DATA_BLOCK "DB_MachineConfig"
{ S7_Optimized_Access := 'TRUE' }
VERSION : 0.1
NON_RETAIN
   VAR
      lastError : Int;
      lastErrorBrand : Int;
      brand { S7_SetPoint := 'False'} : Array[1..16] of "UDT_MachineIOConfig";
   END_VAR


BEGIN
   lastError := 201;
   lastErrorBrand := 2;
   brand[1]."name" := 'Spinner';
   brand[1].cycleArchetype := 1;
   brand[1].in[0].present := TRUE;
   brand[1].in[0].byteOff := 0;
   brand[1].in[0].bitOff := 0;
   brand[1].in[0].inverted := FALSE;
   brand[1].in[1].present := FALSE;
   brand[1].in[1].byteOff := 0;
   brand[1].in[1].bitOff := 0;
   brand[1].in[1].inverted := FALSE;
   brand[1].in[2].present := TRUE;
   brand[1].in[2].byteOff := 0;
   brand[1].in[2].bitOff := 1;
   brand[1].in[2].inverted := FALSE;
   brand[1].in[3].present := TRUE;
   brand[1].in[3].byteOff := 0;
   brand[1].in[3].bitOff := 2;
   brand[1].in[3].inverted := FALSE;
   brand[1].in[4].present := TRUE;
   brand[1].in[4].byteOff := 0;
   brand[1].in[4].bitOff := 3;
   brand[1].in[4].inverted := FALSE;
   brand[1].in[5].present := FALSE;
   brand[1].in[5].byteOff := 0;
   brand[1].in[5].bitOff := 0;
   brand[1].in[5].inverted := FALSE;
   brand[1].in[6].present := TRUE;
   brand[1].in[6].byteOff := 0;
   brand[1].in[6].bitOff := 4;
   brand[1].in[6].inverted := FALSE;
   brand[1].in[7].present := TRUE;
   brand[1].in[7].byteOff := 0;
   brand[1].in[7].bitOff := 5;
   brand[1].in[7].inverted := FALSE;
   brand[1].in[8].present := TRUE;
   brand[1].in[8].byteOff := 0;
   brand[1].in[8].bitOff := 6;
   brand[1].in[8].inverted := FALSE;
   brand[1].in[9].present := FALSE;
   brand[1].in[9].byteOff := 0;
   brand[1].in[9].bitOff := 0;
   brand[1].in[9].inverted := FALSE;
   brand[1].out[0].present := TRUE;
   brand[1].out[0].byteOff := 0;
   brand[1].out[0].bitOff := 0;
   brand[1].out[0].inverted := FALSE;
   brand[1].out[1].present := FALSE;
   brand[1].out[1].byteOff := 0;
   brand[1].out[1].bitOff := 0;
   brand[1].out[1].inverted := FALSE;
   brand[1].out[2].present := TRUE;
   brand[1].out[2].byteOff := 0;
   brand[1].out[2].bitOff := 1;
   brand[1].out[2].inverted := FALSE;
   brand[1].out[3].present := TRUE;
   brand[1].out[3].byteOff := 0;
   brand[1].out[3].bitOff := 2;
   brand[1].out[3].inverted := FALSE;
   brand[1].out[4].present := TRUE;
   brand[1].out[4].byteOff := 0;
   brand[1].out[4].bitOff := 3;
   brand[1].out[4].inverted := FALSE;
   brand[1].out[5].present := FALSE;
   brand[1].out[5].byteOff := 0;
   brand[1].out[5].bitOff := 0;
   brand[1].out[5].inverted := FALSE;
   brand[1].out[6].present := FALSE;
   brand[1].out[6].byteOff := 0;
   brand[1].out[6].bitOff := 0;
   brand[1].out[6].inverted := FALSE;
   brand[1].out[7].present := FALSE;
   brand[1].out[7].byteOff := 0;
   brand[1].out[7].bitOff := 0;
   brand[1].out[7].inverted := FALSE;
   brand[1].out[8].present := TRUE;
   brand[1].out[8].byteOff := 0;
   brand[1].out[8].bitOff := 4;
   brand[1].out[8].inverted := FALSE;
   brand[1].out[9].present := TRUE;
   brand[1].out[9].byteOff := 0;
   brand[1].out[9].bitOff := 5;
   brand[1].out[9].inverted := FALSE;
   brand[1].out[10].present := FALSE;
   brand[1].out[10].byteOff := 0;
   brand[1].out[10].bitOff := 0;
   brand[1].out[10].inverted := FALSE;
   brand[2]."name" := 'HAAS';
   brand[2].cycleArchetype := 2;
   brand[2].in[0].present := TRUE;
   brand[2].in[0].byteOff := 0;
   brand[2].in[0].bitOff := 2;
   brand[2].in[0].inverted := TRUE;
   brand[2].in[1].present := TRUE;
   brand[2].in[1].byteOff := 0;
   brand[2].in[1].bitOff := 2;
   brand[2].in[1].inverted := FALSE;
   brand[2].in[2].present := TRUE;
   brand[2].in[2].byteOff := 0;
   brand[2].in[2].bitOff := 4;
   brand[2].in[2].inverted := FALSE;
   brand[2].in[3].present := TRUE;
   brand[2].in[3].byteOff := 0;
   brand[2].in[3].bitOff := 5;
   brand[2].in[3].inverted := FALSE;
   brand[2].in[4].present := TRUE;
   brand[2].in[4].byteOff := 0;
   brand[2].in[4].bitOff := 6;
   brand[2].in[4].inverted := FALSE;
   brand[2].in[5].present := TRUE;
   brand[2].in[5].byteOff := 0;
   brand[2].in[5].bitOff := 7;
   brand[2].in[5].inverted := FALSE;
   brand[2].in[6].present := TRUE;
   brand[2].in[6].byteOff := 0;
   brand[2].in[6].bitOff := 0;
   brand[2].in[6].inverted := FALSE;
   brand[2].in[7].present := TRUE;
   brand[2].in[7].byteOff := 0;
   brand[2].in[7].bitOff := 1;
   brand[2].in[7].inverted := FALSE;
   brand[2].in[8].present := FALSE;
   brand[2].in[8].byteOff := 0;
   brand[2].in[8].bitOff := 0;
   brand[2].in[8].inverted := FALSE;
   brand[2].in[9].present := FALSE;
   brand[2].in[9].byteOff := 0;
   brand[2].in[9].bitOff := 0;
   brand[2].in[9].inverted := FALSE;
   brand[2].out[0].present := FALSE;
   brand[2].out[0].byteOff := 0;
   brand[2].out[0].bitOff := 0;
   brand[2].out[0].inverted := FALSE;
   brand[2].out[1].present := FALSE;
   brand[2].out[1].byteOff := 0;
   brand[2].out[1].bitOff := 0;
   brand[2].out[1].inverted := FALSE;
   brand[2].out[2].present := TRUE;
   brand[2].out[2].byteOff := 0;
   brand[2].out[2].bitOff := 2;
   brand[2].out[2].inverted := FALSE;
   brand[2].out[3].present := TRUE;
   brand[2].out[3].byteOff := 0;
   brand[2].out[3].bitOff := 3;
   brand[2].out[3].inverted := FALSE;
   brand[2].out[4].present := TRUE;
   brand[2].out[4].byteOff := 0;
   brand[2].out[4].bitOff := 4;
   brand[2].out[4].inverted := FALSE;
   brand[2].out[5].present := TRUE;
   brand[2].out[5].byteOff := 0;
   brand[2].out[5].bitOff := 5;
   brand[2].out[5].inverted := FALSE;
   brand[2].out[6].present := FALSE;
   brand[2].out[6].byteOff := 0;
   brand[2].out[6].bitOff := 0;
   brand[2].out[6].inverted := FALSE;
   brand[2].out[7].present := FALSE;
   brand[2].out[7].byteOff := 0;
   brand[2].out[7].bitOff := 0;
   brand[2].out[7].inverted := FALSE;
   brand[2].out[8].present := TRUE;
   brand[2].out[8].byteOff := 0;
   brand[2].out[8].bitOff := 0;
   brand[2].out[8].inverted := FALSE;
   brand[2].out[9].present := TRUE;
   brand[2].out[9].byteOff := 0;
   brand[2].out[9].bitOff := 6;
   brand[2].out[9].inverted := FALSE;
   brand[2].out[10].present := TRUE;
   brand[2].out[10].byteOff := 0;
   brand[2].out[10].bitOff := 1;
   brand[2].out[10].inverted := FALSE;
   brand[3]."name" := '';
   brand[3].cycleArchetype := 0;
   brand[3].in[0].present := FALSE;
   brand[3].in[0].byteOff := 0;
   brand[3].in[0].bitOff := 0;
   brand[3].in[0].inverted := FALSE;
   brand[3].in[1].present := FALSE;
   brand[3].in[1].byteOff := 0;
   brand[3].in[1].bitOff := 0;
   brand[3].in[1].inverted := FALSE;
   brand[3].in[2].present := FALSE;
   brand[3].in[2].byteOff := 0;
   brand[3].in[2].bitOff := 0;
   brand[3].in[2].inverted := FALSE;
   brand[3].in[3].present := FALSE;
   brand[3].in[3].byteOff := 0;
   brand[3].in[3].bitOff := 0;
   brand[3].in[3].inverted := FALSE;
   brand[3].in[4].present := FALSE;
   brand[3].in[4].byteOff := 0;
   brand[3].in[4].bitOff := 0;
   brand[3].in[4].inverted := FALSE;
   brand[3].in[5].present := FALSE;
   brand[3].in[5].byteOff := 0;
   brand[3].in[5].bitOff := 0;
   brand[3].in[5].inverted := FALSE;
   brand[3].in[6].present := FALSE;
   brand[3].in[6].byteOff := 0;
   brand[3].in[6].bitOff := 0;
   brand[3].in[6].inverted := FALSE;
   brand[3].in[7].present := FALSE;
   brand[3].in[7].byteOff := 0;
   brand[3].in[7].bitOff := 0;
   brand[3].in[7].inverted := FALSE;
   brand[3].in[8].present := FALSE;
   brand[3].in[8].byteOff := 0;
   brand[3].in[8].bitOff := 0;
   brand[3].in[8].inverted := FALSE;
   brand[3].in[9].present := FALSE;
   brand[3].in[9].byteOff := 0;
   brand[3].in[9].bitOff := 0;
   brand[3].in[9].inverted := FALSE;
   brand[3].out[0].present := FALSE;
   brand[3].out[0].byteOff := 0;
   brand[3].out[0].bitOff := 0;
   brand[3].out[0].inverted := FALSE;
   brand[3].out[1].present := FALSE;
   brand[3].out[1].byteOff := 0;
   brand[3].out[1].bitOff := 0;
   brand[3].out[1].inverted := FALSE;
   brand[3].out[2].present := FALSE;
   brand[3].out[2].byteOff := 0;
   brand[3].out[2].bitOff := 0;
   brand[3].out[2].inverted := FALSE;
   brand[3].out[3].present := FALSE;
   brand[3].out[3].byteOff := 0;
   brand[3].out[3].bitOff := 0;
   brand[3].out[3].inverted := FALSE;
   brand[3].out[4].present := FALSE;
   brand[3].out[4].byteOff := 0;
   brand[3].out[4].bitOff := 0;
   brand[3].out[4].inverted := FALSE;
   brand[3].out[5].present := FALSE;
   brand[3].out[5].byteOff := 0;
   brand[3].out[5].bitOff := 0;
   brand[3].out[5].inverted := FALSE;
   brand[3].out[6].present := FALSE;
   brand[3].out[6].byteOff := 0;
   brand[3].out[6].bitOff := 0;
   brand[3].out[6].inverted := FALSE;
   brand[3].out[7].present := FALSE;
   brand[3].out[7].byteOff := 0;
   brand[3].out[7].bitOff := 0;
   brand[3].out[7].inverted := FALSE;
   brand[3].out[8].present := FALSE;
   brand[3].out[8].byteOff := 0;
   brand[3].out[8].bitOff := 0;
   brand[3].out[8].inverted := FALSE;
   brand[3].out[9].present := FALSE;
   brand[3].out[9].byteOff := 0;
   brand[3].out[9].bitOff := 0;
   brand[3].out[9].inverted := FALSE;
   brand[3].out[10].present := FALSE;
   brand[3].out[10].byteOff := 0;
   brand[3].out[10].bitOff := 0;
   brand[3].out[10].inverted := FALSE;
   brand[4]."name" := '';
   brand[4].cycleArchetype := 0;
   brand[4].in[0].present := FALSE;
   brand[4].in[0].byteOff := 0;
   brand[4].in[0].bitOff := 0;
   brand[4].in[0].inverted := FALSE;
   brand[4].in[1].present := FALSE;
   brand[4].in[1].byteOff := 0;
   brand[4].in[1].bitOff := 0;
   brand[4].in[1].inverted := FALSE;
   brand[4].in[2].present := FALSE;
   brand[4].in[2].byteOff := 0;
   brand[4].in[2].bitOff := 0;
   brand[4].in[2].inverted := FALSE;
   brand[4].in[3].present := FALSE;
   brand[4].in[3].byteOff := 0;
   brand[4].in[3].bitOff := 0;
   brand[4].in[3].inverted := FALSE;
   brand[4].in[4].present := FALSE;
   brand[4].in[4].byteOff := 0;
   brand[4].in[4].bitOff := 0;
   brand[4].in[4].inverted := FALSE;
   brand[4].in[5].present := FALSE;
   brand[4].in[5].byteOff := 0;
   brand[4].in[5].bitOff := 0;
   brand[4].in[5].inverted := FALSE;
   brand[4].in[6].present := FALSE;
   brand[4].in[6].byteOff := 0;
   brand[4].in[6].bitOff := 0;
   brand[4].in[6].inverted := FALSE;
   brand[4].in[7].present := FALSE;
   brand[4].in[7].byteOff := 0;
   brand[4].in[7].bitOff := 0;
   brand[4].in[7].inverted := FALSE;
   brand[4].in[8].present := FALSE;
   brand[4].in[8].byteOff := 0;
   brand[4].in[8].bitOff := 0;
   brand[4].in[8].inverted := FALSE;
   brand[4].in[9].present := FALSE;
   brand[4].in[9].byteOff := 0;
   brand[4].in[9].bitOff := 0;
   brand[4].in[9].inverted := FALSE;
   brand[4].out[0].present := FALSE;
   brand[4].out[0].byteOff := 0;
   brand[4].out[0].bitOff := 0;
   brand[4].out[0].inverted := FALSE;
   brand[4].out[1].present := FALSE;
   brand[4].out[1].byteOff := 0;
   brand[4].out[1].bitOff := 0;
   brand[4].out[1].inverted := FALSE;
   brand[4].out[2].present := FALSE;
   brand[4].out[2].byteOff := 0;
   brand[4].out[2].bitOff := 0;
   brand[4].out[2].inverted := FALSE;
   brand[4].out[3].present := FALSE;
   brand[4].out[3].byteOff := 0;
   brand[4].out[3].bitOff := 0;
   brand[4].out[3].inverted := FALSE;
   brand[4].out[4].present := FALSE;
   brand[4].out[4].byteOff := 0;
   brand[4].out[4].bitOff := 0;
   brand[4].out[4].inverted := FALSE;
   brand[4].out[5].present := FALSE;
   brand[4].out[5].byteOff := 0;
   brand[4].out[5].bitOff := 0;
   brand[4].out[5].inverted := FALSE;
   brand[4].out[6].present := FALSE;
   brand[4].out[6].byteOff := 0;
   brand[4].out[6].bitOff := 0;
   brand[4].out[6].inverted := FALSE;
   brand[4].out[7].present := FALSE;
   brand[4].out[7].byteOff := 0;
   brand[4].out[7].bitOff := 0;
   brand[4].out[7].inverted := FALSE;
   brand[4].out[8].present := FALSE;
   brand[4].out[8].byteOff := 0;
   brand[4].out[8].bitOff := 0;
   brand[4].out[8].inverted := FALSE;
   brand[4].out[9].present := FALSE;
   brand[4].out[9].byteOff := 0;
   brand[4].out[9].bitOff := 0;
   brand[4].out[9].inverted := FALSE;
   brand[4].out[10].present := FALSE;
   brand[4].out[10].byteOff := 0;
   brand[4].out[10].bitOff := 0;
   brand[4].out[10].inverted := FALSE;
   brand[5]."name" := '';
   brand[5].cycleArchetype := 0;
   brand[5].in[0].present := FALSE;
   brand[5].in[0].byteOff := 0;
   brand[5].in[0].bitOff := 0;
   brand[5].in[0].inverted := FALSE;
   brand[5].in[1].present := FALSE;
   brand[5].in[1].byteOff := 0;
   brand[5].in[1].bitOff := 0;
   brand[5].in[1].inverted := FALSE;
   brand[5].in[2].present := FALSE;
   brand[5].in[2].byteOff := 0;
   brand[5].in[2].bitOff := 0;
   brand[5].in[2].inverted := FALSE;
   brand[5].in[3].present := FALSE;
   brand[5].in[3].byteOff := 0;
   brand[5].in[3].bitOff := 0;
   brand[5].in[3].inverted := FALSE;
   brand[5].in[4].present := FALSE;
   brand[5].in[4].byteOff := 0;
   brand[5].in[4].bitOff := 0;
   brand[5].in[4].inverted := FALSE;
   brand[5].in[5].present := FALSE;
   brand[5].in[5].byteOff := 0;
   brand[5].in[5].bitOff := 0;
   brand[5].in[5].inverted := FALSE;
   brand[5].in[6].present := FALSE;
   brand[5].in[6].byteOff := 0;
   brand[5].in[6].bitOff := 0;
   brand[5].in[6].inverted := FALSE;
   brand[5].in[7].present := FALSE;
   brand[5].in[7].byteOff := 0;
   brand[5].in[7].bitOff := 0;
   brand[5].in[7].inverted := FALSE;
   brand[5].in[8].present := FALSE;
   brand[5].in[8].byteOff := 0;
   brand[5].in[8].bitOff := 0;
   brand[5].in[8].inverted := FALSE;
   brand[5].in[9].present := FALSE;
   brand[5].in[9].byteOff := 0;
   brand[5].in[9].bitOff := 0;
   brand[5].in[9].inverted := FALSE;
   brand[5].out[0].present := FALSE;
   brand[5].out[0].byteOff := 0;
   brand[5].out[0].bitOff := 0;
   brand[5].out[0].inverted := FALSE;
   brand[5].out[1].present := FALSE;
   brand[5].out[1].byteOff := 0;
   brand[5].out[1].bitOff := 0;
   brand[5].out[1].inverted := FALSE;
   brand[5].out[2].present := FALSE;
   brand[5].out[2].byteOff := 0;
   brand[5].out[2].bitOff := 0;
   brand[5].out[2].inverted := FALSE;
   brand[5].out[3].present := FALSE;
   brand[5].out[3].byteOff := 0;
   brand[5].out[3].bitOff := 0;
   brand[5].out[3].inverted := FALSE;
   brand[5].out[4].present := FALSE;
   brand[5].out[4].byteOff := 0;
   brand[5].out[4].bitOff := 0;
   brand[5].out[4].inverted := FALSE;
   brand[5].out[5].present := FALSE;
   brand[5].out[5].byteOff := 0;
   brand[5].out[5].bitOff := 0;
   brand[5].out[5].inverted := FALSE;
   brand[5].out[6].present := FALSE;
   brand[5].out[6].byteOff := 0;
   brand[5].out[6].bitOff := 0;
   brand[5].out[6].inverted := FALSE;
   brand[5].out[7].present := FALSE;
   brand[5].out[7].byteOff := 0;
   brand[5].out[7].bitOff := 0;
   brand[5].out[7].inverted := FALSE;
   brand[5].out[8].present := FALSE;
   brand[5].out[8].byteOff := 0;
   brand[5].out[8].bitOff := 0;
   brand[5].out[8].inverted := FALSE;
   brand[5].out[9].present := FALSE;
   brand[5].out[9].byteOff := 0;
   brand[5].out[9].bitOff := 0;
   brand[5].out[9].inverted := FALSE;
   brand[5].out[10].present := FALSE;
   brand[5].out[10].byteOff := 0;
   brand[5].out[10].bitOff := 0;
   brand[5].out[10].inverted := FALSE;
   brand[6]."name" := '';
   brand[6].cycleArchetype := 0;
   brand[6].in[0].present := FALSE;
   brand[6].in[0].byteOff := 0;
   brand[6].in[0].bitOff := 0;
   brand[6].in[0].inverted := FALSE;
   brand[6].in[1].present := FALSE;
   brand[6].in[1].byteOff := 0;
   brand[6].in[1].bitOff := 0;
   brand[6].in[1].inverted := FALSE;
   brand[6].in[2].present := FALSE;
   brand[6].in[2].byteOff := 0;
   brand[6].in[2].bitOff := 0;
   brand[6].in[2].inverted := FALSE;
   brand[6].in[3].present := FALSE;
   brand[6].in[3].byteOff := 0;
   brand[6].in[3].bitOff := 0;
   brand[6].in[3].inverted := FALSE;
   brand[6].in[4].present := FALSE;
   brand[6].in[4].byteOff := 0;
   brand[6].in[4].bitOff := 0;
   brand[6].in[4].inverted := FALSE;
   brand[6].in[5].present := FALSE;
   brand[6].in[5].byteOff := 0;
   brand[6].in[5].bitOff := 0;
   brand[6].in[5].inverted := FALSE;
   brand[6].in[6].present := FALSE;
   brand[6].in[6].byteOff := 0;
   brand[6].in[6].bitOff := 0;
   brand[6].in[6].inverted := FALSE;
   brand[6].in[7].present := FALSE;
   brand[6].in[7].byteOff := 0;
   brand[6].in[7].bitOff := 0;
   brand[6].in[7].inverted := FALSE;
   brand[6].in[8].present := FALSE;
   brand[6].in[8].byteOff := 0;
   brand[6].in[8].bitOff := 0;
   brand[6].in[8].inverted := FALSE;
   brand[6].in[9].present := FALSE;
   brand[6].in[9].byteOff := 0;
   brand[6].in[9].bitOff := 0;
   brand[6].in[9].inverted := FALSE;
   brand[6].out[0].present := FALSE;
   brand[6].out[0].byteOff := 0;
   brand[6].out[0].bitOff := 0;
   brand[6].out[0].inverted := FALSE;
   brand[6].out[1].present := FALSE;
   brand[6].out[1].byteOff := 0;
   brand[6].out[1].bitOff := 0;
   brand[6].out[1].inverted := FALSE;
   brand[6].out[2].present := FALSE;
   brand[6].out[2].byteOff := 0;
   brand[6].out[2].bitOff := 0;
   brand[6].out[2].inverted := FALSE;
   brand[6].out[3].present := FALSE;
   brand[6].out[3].byteOff := 0;
   brand[6].out[3].bitOff := 0;
   brand[6].out[3].inverted := FALSE;
   brand[6].out[4].present := FALSE;
   brand[6].out[4].byteOff := 0;
   brand[6].out[4].bitOff := 0;
   brand[6].out[4].inverted := FALSE;
   brand[6].out[5].present := FALSE;
   brand[6].out[5].byteOff := 0;
   brand[6].out[5].bitOff := 0;
   brand[6].out[5].inverted := FALSE;
   brand[6].out[6].present := FALSE;
   brand[6].out[6].byteOff := 0;
   brand[6].out[6].bitOff := 0;
   brand[6].out[6].inverted := FALSE;
   brand[6].out[7].present := FALSE;
   brand[6].out[7].byteOff := 0;
   brand[6].out[7].bitOff := 0;
   brand[6].out[7].inverted := FALSE;
   brand[6].out[8].present := FALSE;
   brand[6].out[8].byteOff := 0;
   brand[6].out[8].bitOff := 0;
   brand[6].out[8].inverted := FALSE;
   brand[6].out[9].present := FALSE;
   brand[6].out[9].byteOff := 0;
   brand[6].out[9].bitOff := 0;
   brand[6].out[9].inverted := FALSE;
   brand[6].out[10].present := FALSE;
   brand[6].out[10].byteOff := 0;
   brand[6].out[10].bitOff := 0;
   brand[6].out[10].inverted := FALSE;
   brand[7]."name" := '';
   brand[7].cycleArchetype := 0;
   brand[7].in[0].present := FALSE;
   brand[7].in[0].byteOff := 0;
   brand[7].in[0].bitOff := 0;
   brand[7].in[0].inverted := FALSE;
   brand[7].in[1].present := FALSE;
   brand[7].in[1].byteOff := 0;
   brand[7].in[1].bitOff := 0;
   brand[7].in[1].inverted := FALSE;
   brand[7].in[2].present := FALSE;
   brand[7].in[2].byteOff := 0;
   brand[7].in[2].bitOff := 0;
   brand[7].in[2].inverted := FALSE;
   brand[7].in[3].present := FALSE;
   brand[7].in[3].byteOff := 0;
   brand[7].in[3].bitOff := 0;
   brand[7].in[3].inverted := FALSE;
   brand[7].in[4].present := FALSE;
   brand[7].in[4].byteOff := 0;
   brand[7].in[4].bitOff := 0;
   brand[7].in[4].inverted := FALSE;
   brand[7].in[5].present := FALSE;
   brand[7].in[5].byteOff := 0;
   brand[7].in[5].bitOff := 0;
   brand[7].in[5].inverted := FALSE;
   brand[7].in[6].present := FALSE;
   brand[7].in[6].byteOff := 0;
   brand[7].in[6].bitOff := 0;
   brand[7].in[6].inverted := FALSE;
   brand[7].in[7].present := FALSE;
   brand[7].in[7].byteOff := 0;
   brand[7].in[7].bitOff := 0;
   brand[7].in[7].inverted := FALSE;
   brand[7].in[8].present := FALSE;
   brand[7].in[8].byteOff := 0;
   brand[7].in[8].bitOff := 0;
   brand[7].in[8].inverted := FALSE;
   brand[7].in[9].present := FALSE;
   brand[7].in[9].byteOff := 0;
   brand[7].in[9].bitOff := 0;
   brand[7].in[9].inverted := FALSE;
   brand[7].out[0].present := FALSE;
   brand[7].out[0].byteOff := 0;
   brand[7].out[0].bitOff := 0;
   brand[7].out[0].inverted := FALSE;
   brand[7].out[1].present := FALSE;
   brand[7].out[1].byteOff := 0;
   brand[7].out[1].bitOff := 0;
   brand[7].out[1].inverted := FALSE;
   brand[7].out[2].present := FALSE;
   brand[7].out[2].byteOff := 0;
   brand[7].out[2].bitOff := 0;
   brand[7].out[2].inverted := FALSE;
   brand[7].out[3].present := FALSE;
   brand[7].out[3].byteOff := 0;
   brand[7].out[3].bitOff := 0;
   brand[7].out[3].inverted := FALSE;
   brand[7].out[4].present := FALSE;
   brand[7].out[4].byteOff := 0;
   brand[7].out[4].bitOff := 0;
   brand[7].out[4].inverted := FALSE;
   brand[7].out[5].present := FALSE;
   brand[7].out[5].byteOff := 0;
   brand[7].out[5].bitOff := 0;
   brand[7].out[5].inverted := FALSE;
   brand[7].out[6].present := FALSE;
   brand[7].out[6].byteOff := 0;
   brand[7].out[6].bitOff := 0;
   brand[7].out[6].inverted := FALSE;
   brand[7].out[7].present := FALSE;
   brand[7].out[7].byteOff := 0;
   brand[7].out[7].bitOff := 0;
   brand[7].out[7].inverted := FALSE;
   brand[7].out[8].present := FALSE;
   brand[7].out[8].byteOff := 0;
   brand[7].out[8].bitOff := 0;
   brand[7].out[8].inverted := FALSE;
   brand[7].out[9].present := FALSE;
   brand[7].out[9].byteOff := 0;
   brand[7].out[9].bitOff := 0;
   brand[7].out[9].inverted := FALSE;
   brand[7].out[10].present := FALSE;
   brand[7].out[10].byteOff := 0;
   brand[7].out[10].bitOff := 0;
   brand[7].out[10].inverted := FALSE;
   brand[8]."name" := '';
   brand[8].cycleArchetype := 0;
   brand[8].in[0].present := FALSE;
   brand[8].in[0].byteOff := 0;
   brand[8].in[0].bitOff := 0;
   brand[8].in[0].inverted := FALSE;
   brand[8].in[1].present := FALSE;
   brand[8].in[1].byteOff := 0;
   brand[8].in[1].bitOff := 0;
   brand[8].in[1].inverted := FALSE;
   brand[8].in[2].present := FALSE;
   brand[8].in[2].byteOff := 0;
   brand[8].in[2].bitOff := 0;
   brand[8].in[2].inverted := FALSE;
   brand[8].in[3].present := FALSE;
   brand[8].in[3].byteOff := 0;
   brand[8].in[3].bitOff := 0;
   brand[8].in[3].inverted := FALSE;
   brand[8].in[4].present := FALSE;
   brand[8].in[4].byteOff := 0;
   brand[8].in[4].bitOff := 0;
   brand[8].in[4].inverted := FALSE;
   brand[8].in[5].present := FALSE;
   brand[8].in[5].byteOff := 0;
   brand[8].in[5].bitOff := 0;
   brand[8].in[5].inverted := FALSE;
   brand[8].in[6].present := FALSE;
   brand[8].in[6].byteOff := 0;
   brand[8].in[6].bitOff := 0;
   brand[8].in[6].inverted := FALSE;
   brand[8].in[7].present := FALSE;
   brand[8].in[7].byteOff := 0;
   brand[8].in[7].bitOff := 0;
   brand[8].in[7].inverted := FALSE;
   brand[8].in[8].present := FALSE;
   brand[8].in[8].byteOff := 0;
   brand[8].in[8].bitOff := 0;
   brand[8].in[8].inverted := FALSE;
   brand[8].in[9].present := FALSE;
   brand[8].in[9].byteOff := 0;
   brand[8].in[9].bitOff := 0;
   brand[8].in[9].inverted := FALSE;
   brand[8].out[0].present := FALSE;
   brand[8].out[0].byteOff := 0;
   brand[8].out[0].bitOff := 0;
   brand[8].out[0].inverted := FALSE;
   brand[8].out[1].present := FALSE;
   brand[8].out[1].byteOff := 0;
   brand[8].out[1].bitOff := 0;
   brand[8].out[1].inverted := FALSE;
   brand[8].out[2].present := FALSE;
   brand[8].out[2].byteOff := 0;
   brand[8].out[2].bitOff := 0;
   brand[8].out[2].inverted := FALSE;
   brand[8].out[3].present := FALSE;
   brand[8].out[3].byteOff := 0;
   brand[8].out[3].bitOff := 0;
   brand[8].out[3].inverted := FALSE;
   brand[8].out[4].present := FALSE;
   brand[8].out[4].byteOff := 0;
   brand[8].out[4].bitOff := 0;
   brand[8].out[4].inverted := FALSE;
   brand[8].out[5].present := FALSE;
   brand[8].out[5].byteOff := 0;
   brand[8].out[5].bitOff := 0;
   brand[8].out[5].inverted := FALSE;
   brand[8].out[6].present := FALSE;
   brand[8].out[6].byteOff := 0;
   brand[8].out[6].bitOff := 0;
   brand[8].out[6].inverted := FALSE;
   brand[8].out[7].present := FALSE;
   brand[8].out[7].byteOff := 0;
   brand[8].out[7].bitOff := 0;
   brand[8].out[7].inverted := FALSE;
   brand[8].out[8].present := FALSE;
   brand[8].out[8].byteOff := 0;
   brand[8].out[8].bitOff := 0;
   brand[8].out[8].inverted := FALSE;
   brand[8].out[9].present := FALSE;
   brand[8].out[9].byteOff := 0;
   brand[8].out[9].bitOff := 0;
   brand[8].out[9].inverted := FALSE;
   brand[8].out[10].present := FALSE;
   brand[8].out[10].byteOff := 0;
   brand[8].out[10].bitOff := 0;
   brand[8].out[10].inverted := FALSE;
   brand[9]."name" := '';
   brand[9].cycleArchetype := 0;
   brand[9].in[0].present := FALSE;
   brand[9].in[0].byteOff := 0;
   brand[9].in[0].bitOff := 0;
   brand[9].in[0].inverted := FALSE;
   brand[9].in[1].present := FALSE;
   brand[9].in[1].byteOff := 0;
   brand[9].in[1].bitOff := 0;
   brand[9].in[1].inverted := FALSE;
   brand[9].in[2].present := FALSE;
   brand[9].in[2].byteOff := 0;
   brand[9].in[2].bitOff := 0;
   brand[9].in[2].inverted := FALSE;
   brand[9].in[3].present := FALSE;
   brand[9].in[3].byteOff := 0;
   brand[9].in[3].bitOff := 0;
   brand[9].in[3].inverted := FALSE;
   brand[9].in[4].present := FALSE;
   brand[9].in[4].byteOff := 0;
   brand[9].in[4].bitOff := 0;
   brand[9].in[4].inverted := FALSE;
   brand[9].in[5].present := FALSE;
   brand[9].in[5].byteOff := 0;
   brand[9].in[5].bitOff := 0;
   brand[9].in[5].inverted := FALSE;
   brand[9].in[6].present := FALSE;
   brand[9].in[6].byteOff := 0;
   brand[9].in[6].bitOff := 0;
   brand[9].in[6].inverted := FALSE;
   brand[9].in[7].present := FALSE;
   brand[9].in[7].byteOff := 0;
   brand[9].in[7].bitOff := 0;
   brand[9].in[7].inverted := FALSE;
   brand[9].in[8].present := FALSE;
   brand[9].in[8].byteOff := 0;
   brand[9].in[8].bitOff := 0;
   brand[9].in[8].inverted := FALSE;
   brand[9].in[9].present := FALSE;
   brand[9].in[9].byteOff := 0;
   brand[9].in[9].bitOff := 0;
   brand[9].in[9].inverted := FALSE;
   brand[9].out[0].present := FALSE;
   brand[9].out[0].byteOff := 0;
   brand[9].out[0].bitOff := 0;
   brand[9].out[0].inverted := FALSE;
   brand[9].out[1].present := FALSE;
   brand[9].out[1].byteOff := 0;
   brand[9].out[1].bitOff := 0;
   brand[9].out[1].inverted := FALSE;
   brand[9].out[2].present := FALSE;
   brand[9].out[2].byteOff := 0;
   brand[9].out[2].bitOff := 0;
   brand[9].out[2].inverted := FALSE;
   brand[9].out[3].present := FALSE;
   brand[9].out[3].byteOff := 0;
   brand[9].out[3].bitOff := 0;
   brand[9].out[3].inverted := FALSE;
   brand[9].out[4].present := FALSE;
   brand[9].out[4].byteOff := 0;
   brand[9].out[4].bitOff := 0;
   brand[9].out[4].inverted := FALSE;
   brand[9].out[5].present := FALSE;
   brand[9].out[5].byteOff := 0;
   brand[9].out[5].bitOff := 0;
   brand[9].out[5].inverted := FALSE;
   brand[9].out[6].present := FALSE;
   brand[9].out[6].byteOff := 0;
   brand[9].out[6].bitOff := 0;
   brand[9].out[6].inverted := FALSE;
   brand[9].out[7].present := FALSE;
   brand[9].out[7].byteOff := 0;
   brand[9].out[7].bitOff := 0;
   brand[9].out[7].inverted := FALSE;
   brand[9].out[8].present := FALSE;
   brand[9].out[8].byteOff := 0;
   brand[9].out[8].bitOff := 0;
   brand[9].out[8].inverted := FALSE;
   brand[9].out[9].present := FALSE;
   brand[9].out[9].byteOff := 0;
   brand[9].out[9].bitOff := 0;
   brand[9].out[9].inverted := FALSE;
   brand[9].out[10].present := FALSE;
   brand[9].out[10].byteOff := 0;
   brand[9].out[10].bitOff := 0;
   brand[9].out[10].inverted := FALSE;
   brand[10]."name" := '';
   brand[10].cycleArchetype := 0;
   brand[10].in[0].present := FALSE;
   brand[10].in[0].byteOff := 0;
   brand[10].in[0].bitOff := 0;
   brand[10].in[0].inverted := FALSE;
   brand[10].in[1].present := FALSE;
   brand[10].in[1].byteOff := 0;
   brand[10].in[1].bitOff := 0;
   brand[10].in[1].inverted := FALSE;
   brand[10].in[2].present := FALSE;
   brand[10].in[2].byteOff := 0;
   brand[10].in[2].bitOff := 0;
   brand[10].in[2].inverted := FALSE;
   brand[10].in[3].present := FALSE;
   brand[10].in[3].byteOff := 0;
   brand[10].in[3].bitOff := 0;
   brand[10].in[3].inverted := FALSE;
   brand[10].in[4].present := FALSE;
   brand[10].in[4].byteOff := 0;
   brand[10].in[4].bitOff := 0;
   brand[10].in[4].inverted := FALSE;
   brand[10].in[5].present := FALSE;
   brand[10].in[5].byteOff := 0;
   brand[10].in[5].bitOff := 0;
   brand[10].in[5].inverted := FALSE;
   brand[10].in[6].present := FALSE;
   brand[10].in[6].byteOff := 0;
   brand[10].in[6].bitOff := 0;
   brand[10].in[6].inverted := FALSE;
   brand[10].in[7].present := FALSE;
   brand[10].in[7].byteOff := 0;
   brand[10].in[7].bitOff := 0;
   brand[10].in[7].inverted := FALSE;
   brand[10].in[8].present := FALSE;
   brand[10].in[8].byteOff := 0;
   brand[10].in[8].bitOff := 0;
   brand[10].in[8].inverted := FALSE;
   brand[10].in[9].present := FALSE;
   brand[10].in[9].byteOff := 0;
   brand[10].in[9].bitOff := 0;
   brand[10].in[9].inverted := FALSE;
   brand[10].out[0].present := FALSE;
   brand[10].out[0].byteOff := 0;
   brand[10].out[0].bitOff := 0;
   brand[10].out[0].inverted := FALSE;
   brand[10].out[1].present := FALSE;
   brand[10].out[1].byteOff := 0;
   brand[10].out[1].bitOff := 0;
   brand[10].out[1].inverted := FALSE;
   brand[10].out[2].present := FALSE;
   brand[10].out[2].byteOff := 0;
   brand[10].out[2].bitOff := 0;
   brand[10].out[2].inverted := FALSE;
   brand[10].out[3].present := FALSE;
   brand[10].out[3].byteOff := 0;
   brand[10].out[3].bitOff := 0;
   brand[10].out[3].inverted := FALSE;
   brand[10].out[4].present := FALSE;
   brand[10].out[4].byteOff := 0;
   brand[10].out[4].bitOff := 0;
   brand[10].out[4].inverted := FALSE;
   brand[10].out[5].present := FALSE;
   brand[10].out[5].byteOff := 0;
   brand[10].out[5].bitOff := 0;
   brand[10].out[5].inverted := FALSE;
   brand[10].out[6].present := FALSE;
   brand[10].out[6].byteOff := 0;
   brand[10].out[6].bitOff := 0;
   brand[10].out[6].inverted := FALSE;
   brand[10].out[7].present := FALSE;
   brand[10].out[7].byteOff := 0;
   brand[10].out[7].bitOff := 0;
   brand[10].out[7].inverted := FALSE;
   brand[10].out[8].present := FALSE;
   brand[10].out[8].byteOff := 0;
   brand[10].out[8].bitOff := 0;
   brand[10].out[8].inverted := FALSE;
   brand[10].out[9].present := FALSE;
   brand[10].out[9].byteOff := 0;
   brand[10].out[9].bitOff := 0;
   brand[10].out[9].inverted := FALSE;
   brand[10].out[10].present := FALSE;
   brand[10].out[10].byteOff := 0;
   brand[10].out[10].bitOff := 0;
   brand[10].out[10].inverted := FALSE;
   brand[11]."name" := '';
   brand[11].cycleArchetype := 0;
   brand[11].in[0].present := FALSE;
   brand[11].in[0].byteOff := 0;
   brand[11].in[0].bitOff := 0;
   brand[11].in[0].inverted := FALSE;
   brand[11].in[1].present := FALSE;
   brand[11].in[1].byteOff := 0;
   brand[11].in[1].bitOff := 0;
   brand[11].in[1].inverted := FALSE;
   brand[11].in[2].present := FALSE;
   brand[11].in[2].byteOff := 0;
   brand[11].in[2].bitOff := 0;
   brand[11].in[2].inverted := FALSE;
   brand[11].in[3].present := FALSE;
   brand[11].in[3].byteOff := 0;
   brand[11].in[3].bitOff := 0;
   brand[11].in[3].inverted := FALSE;
   brand[11].in[4].present := FALSE;
   brand[11].in[4].byteOff := 0;
   brand[11].in[4].bitOff := 0;
   brand[11].in[4].inverted := FALSE;
   brand[11].in[5].present := FALSE;
   brand[11].in[5].byteOff := 0;
   brand[11].in[5].bitOff := 0;
   brand[11].in[5].inverted := FALSE;
   brand[11].in[6].present := FALSE;
   brand[11].in[6].byteOff := 0;
   brand[11].in[6].bitOff := 0;
   brand[11].in[6].inverted := FALSE;
   brand[11].in[7].present := FALSE;
   brand[11].in[7].byteOff := 0;
   brand[11].in[7].bitOff := 0;
   brand[11].in[7].inverted := FALSE;
   brand[11].in[8].present := FALSE;
   brand[11].in[8].byteOff := 0;
   brand[11].in[8].bitOff := 0;
   brand[11].in[8].inverted := FALSE;
   brand[11].in[9].present := FALSE;
   brand[11].in[9].byteOff := 0;
   brand[11].in[9].bitOff := 0;
   brand[11].in[9].inverted := FALSE;
   brand[11].out[0].present := FALSE;
   brand[11].out[0].byteOff := 0;
   brand[11].out[0].bitOff := 0;
   brand[11].out[0].inverted := FALSE;
   brand[11].out[1].present := FALSE;
   brand[11].out[1].byteOff := 0;
   brand[11].out[1].bitOff := 0;
   brand[11].out[1].inverted := FALSE;
   brand[11].out[2].present := FALSE;
   brand[11].out[2].byteOff := 0;
   brand[11].out[2].bitOff := 0;
   brand[11].out[2].inverted := FALSE;
   brand[11].out[3].present := FALSE;
   brand[11].out[3].byteOff := 0;
   brand[11].out[3].bitOff := 0;
   brand[11].out[3].inverted := FALSE;
   brand[11].out[4].present := FALSE;
   brand[11].out[4].byteOff := 0;
   brand[11].out[4].bitOff := 0;
   brand[11].out[4].inverted := FALSE;
   brand[11].out[5].present := FALSE;
   brand[11].out[5].byteOff := 0;
   brand[11].out[5].bitOff := 0;
   brand[11].out[5].inverted := FALSE;
   brand[11].out[6].present := FALSE;
   brand[11].out[6].byteOff := 0;
   brand[11].out[6].bitOff := 0;
   brand[11].out[6].inverted := FALSE;
   brand[11].out[7].present := FALSE;
   brand[11].out[7].byteOff := 0;
   brand[11].out[7].bitOff := 0;
   brand[11].out[7].inverted := FALSE;
   brand[11].out[8].present := FALSE;
   brand[11].out[8].byteOff := 0;
   brand[11].out[8].bitOff := 0;
   brand[11].out[8].inverted := FALSE;
   brand[11].out[9].present := FALSE;
   brand[11].out[9].byteOff := 0;
   brand[11].out[9].bitOff := 0;
   brand[11].out[9].inverted := FALSE;
   brand[11].out[10].present := FALSE;
   brand[11].out[10].byteOff := 0;
   brand[11].out[10].bitOff := 0;
   brand[11].out[10].inverted := FALSE;
   brand[12]."name" := '';
   brand[12].cycleArchetype := 0;
   brand[12].in[0].present := FALSE;
   brand[12].in[0].byteOff := 0;
   brand[12].in[0].bitOff := 0;
   brand[12].in[0].inverted := FALSE;
   brand[12].in[1].present := FALSE;
   brand[12].in[1].byteOff := 0;
   brand[12].in[1].bitOff := 0;
   brand[12].in[1].inverted := FALSE;
   brand[12].in[2].present := FALSE;
   brand[12].in[2].byteOff := 0;
   brand[12].in[2].bitOff := 0;
   brand[12].in[2].inverted := FALSE;
   brand[12].in[3].present := FALSE;
   brand[12].in[3].byteOff := 0;
   brand[12].in[3].bitOff := 0;
   brand[12].in[3].inverted := FALSE;
   brand[12].in[4].present := FALSE;
   brand[12].in[4].byteOff := 0;
   brand[12].in[4].bitOff := 0;
   brand[12].in[4].inverted := FALSE;
   brand[12].in[5].present := FALSE;
   brand[12].in[5].byteOff := 0;
   brand[12].in[5].bitOff := 0;
   brand[12].in[5].inverted := FALSE;
   brand[12].in[6].present := FALSE;
   brand[12].in[6].byteOff := 0;
   brand[12].in[6].bitOff := 0;
   brand[12].in[6].inverted := FALSE;
   brand[12].in[7].present := FALSE;
   brand[12].in[7].byteOff := 0;
   brand[12].in[7].bitOff := 0;
   brand[12].in[7].inverted := FALSE;
   brand[12].in[8].present := FALSE;
   brand[12].in[8].byteOff := 0;
   brand[12].in[8].bitOff := 0;
   brand[12].in[8].inverted := FALSE;
   brand[12].in[9].present := FALSE;
   brand[12].in[9].byteOff := 0;
   brand[12].in[9].bitOff := 0;
   brand[12].in[9].inverted := FALSE;
   brand[12].out[0].present := FALSE;
   brand[12].out[0].byteOff := 0;
   brand[12].out[0].bitOff := 0;
   brand[12].out[0].inverted := FALSE;
   brand[12].out[1].present := FALSE;
   brand[12].out[1].byteOff := 0;
   brand[12].out[1].bitOff := 0;
   brand[12].out[1].inverted := FALSE;
   brand[12].out[2].present := FALSE;
   brand[12].out[2].byteOff := 0;
   brand[12].out[2].bitOff := 0;
   brand[12].out[2].inverted := FALSE;
   brand[12].out[3].present := FALSE;
   brand[12].out[3].byteOff := 0;
   brand[12].out[3].bitOff := 0;
   brand[12].out[3].inverted := FALSE;
   brand[12].out[4].present := FALSE;
   brand[12].out[4].byteOff := 0;
   brand[12].out[4].bitOff := 0;
   brand[12].out[4].inverted := FALSE;
   brand[12].out[5].present := FALSE;
   brand[12].out[5].byteOff := 0;
   brand[12].out[5].bitOff := 0;
   brand[12].out[5].inverted := FALSE;
   brand[12].out[6].present := FALSE;
   brand[12].out[6].byteOff := 0;
   brand[12].out[6].bitOff := 0;
   brand[12].out[6].inverted := FALSE;
   brand[12].out[7].present := FALSE;
   brand[12].out[7].byteOff := 0;
   brand[12].out[7].bitOff := 0;
   brand[12].out[7].inverted := FALSE;
   brand[12].out[8].present := FALSE;
   brand[12].out[8].byteOff := 0;
   brand[12].out[8].bitOff := 0;
   brand[12].out[8].inverted := FALSE;
   brand[12].out[9].present := FALSE;
   brand[12].out[9].byteOff := 0;
   brand[12].out[9].bitOff := 0;
   brand[12].out[9].inverted := FALSE;
   brand[12].out[10].present := FALSE;
   brand[12].out[10].byteOff := 0;
   brand[12].out[10].bitOff := 0;
   brand[12].out[10].inverted := FALSE;
   brand[13]."name" := '';
   brand[13].cycleArchetype := 0;
   brand[13].in[0].present := FALSE;
   brand[13].in[0].byteOff := 0;
   brand[13].in[0].bitOff := 0;
   brand[13].in[0].inverted := FALSE;
   brand[13].in[1].present := FALSE;
   brand[13].in[1].byteOff := 0;
   brand[13].in[1].bitOff := 0;
   brand[13].in[1].inverted := FALSE;
   brand[13].in[2].present := FALSE;
   brand[13].in[2].byteOff := 0;
   brand[13].in[2].bitOff := 0;
   brand[13].in[2].inverted := FALSE;
   brand[13].in[3].present := FALSE;
   brand[13].in[3].byteOff := 0;
   brand[13].in[3].bitOff := 0;
   brand[13].in[3].inverted := FALSE;
   brand[13].in[4].present := FALSE;
   brand[13].in[4].byteOff := 0;
   brand[13].in[4].bitOff := 0;
   brand[13].in[4].inverted := FALSE;
   brand[13].in[5].present := FALSE;
   brand[13].in[5].byteOff := 0;
   brand[13].in[5].bitOff := 0;
   brand[13].in[5].inverted := FALSE;
   brand[13].in[6].present := FALSE;
   brand[13].in[6].byteOff := 0;
   brand[13].in[6].bitOff := 0;
   brand[13].in[6].inverted := FALSE;
   brand[13].in[7].present := FALSE;
   brand[13].in[7].byteOff := 0;
   brand[13].in[7].bitOff := 0;
   brand[13].in[7].inverted := FALSE;
   brand[13].in[8].present := FALSE;
   brand[13].in[8].byteOff := 0;
   brand[13].in[8].bitOff := 0;
   brand[13].in[8].inverted := FALSE;
   brand[13].in[9].present := FALSE;
   brand[13].in[9].byteOff := 0;
   brand[13].in[9].bitOff := 0;
   brand[13].in[9].inverted := FALSE;
   brand[13].out[0].present := FALSE;
   brand[13].out[0].byteOff := 0;
   brand[13].out[0].bitOff := 0;
   brand[13].out[0].inverted := FALSE;
   brand[13].out[1].present := FALSE;
   brand[13].out[1].byteOff := 0;
   brand[13].out[1].bitOff := 0;
   brand[13].out[1].inverted := FALSE;
   brand[13].out[2].present := FALSE;
   brand[13].out[2].byteOff := 0;
   brand[13].out[2].bitOff := 0;
   brand[13].out[2].inverted := FALSE;
   brand[13].out[3].present := FALSE;
   brand[13].out[3].byteOff := 0;
   brand[13].out[3].bitOff := 0;
   brand[13].out[3].inverted := FALSE;
   brand[13].out[4].present := FALSE;
   brand[13].out[4].byteOff := 0;
   brand[13].out[4].bitOff := 0;
   brand[13].out[4].inverted := FALSE;
   brand[13].out[5].present := FALSE;
   brand[13].out[5].byteOff := 0;
   brand[13].out[5].bitOff := 0;
   brand[13].out[5].inverted := FALSE;
   brand[13].out[6].present := FALSE;
   brand[13].out[6].byteOff := 0;
   brand[13].out[6].bitOff := 0;
   brand[13].out[6].inverted := FALSE;
   brand[13].out[7].present := FALSE;
   brand[13].out[7].byteOff := 0;
   brand[13].out[7].bitOff := 0;
   brand[13].out[7].inverted := FALSE;
   brand[13].out[8].present := FALSE;
   brand[13].out[8].byteOff := 0;
   brand[13].out[8].bitOff := 0;
   brand[13].out[8].inverted := FALSE;
   brand[13].out[9].present := FALSE;
   brand[13].out[9].byteOff := 0;
   brand[13].out[9].bitOff := 0;
   brand[13].out[9].inverted := FALSE;
   brand[13].out[10].present := FALSE;
   brand[13].out[10].byteOff := 0;
   brand[13].out[10].bitOff := 0;
   brand[13].out[10].inverted := FALSE;
   brand[14]."name" := '';
   brand[14].cycleArchetype := 0;
   brand[14].in[0].present := FALSE;
   brand[14].in[0].byteOff := 0;
   brand[14].in[0].bitOff := 0;
   brand[14].in[0].inverted := FALSE;
   brand[14].in[1].present := FALSE;
   brand[14].in[1].byteOff := 0;
   brand[14].in[1].bitOff := 0;
   brand[14].in[1].inverted := FALSE;
   brand[14].in[2].present := FALSE;
   brand[14].in[2].byteOff := 0;
   brand[14].in[2].bitOff := 0;
   brand[14].in[2].inverted := FALSE;
   brand[14].in[3].present := FALSE;
   brand[14].in[3].byteOff := 0;
   brand[14].in[3].bitOff := 0;
   brand[14].in[3].inverted := FALSE;
   brand[14].in[4].present := FALSE;
   brand[14].in[4].byteOff := 0;
   brand[14].in[4].bitOff := 0;
   brand[14].in[4].inverted := FALSE;
   brand[14].in[5].present := FALSE;
   brand[14].in[5].byteOff := 0;
   brand[14].in[5].bitOff := 0;
   brand[14].in[5].inverted := FALSE;
   brand[14].in[6].present := FALSE;
   brand[14].in[6].byteOff := 0;
   brand[14].in[6].bitOff := 0;
   brand[14].in[6].inverted := FALSE;
   brand[14].in[7].present := FALSE;
   brand[14].in[7].byteOff := 0;
   brand[14].in[7].bitOff := 0;
   brand[14].in[7].inverted := FALSE;
   brand[14].in[8].present := FALSE;
   brand[14].in[8].byteOff := 0;
   brand[14].in[8].bitOff := 0;
   brand[14].in[8].inverted := FALSE;
   brand[14].in[9].present := FALSE;
   brand[14].in[9].byteOff := 0;
   brand[14].in[9].bitOff := 0;
   brand[14].in[9].inverted := FALSE;
   brand[14].out[0].present := FALSE;
   brand[14].out[0].byteOff := 0;
   brand[14].out[0].bitOff := 0;
   brand[14].out[0].inverted := FALSE;
   brand[14].out[1].present := FALSE;
   brand[14].out[1].byteOff := 0;
   brand[14].out[1].bitOff := 0;
   brand[14].out[1].inverted := FALSE;
   brand[14].out[2].present := FALSE;
   brand[14].out[2].byteOff := 0;
   brand[14].out[2].bitOff := 0;
   brand[14].out[2].inverted := FALSE;
   brand[14].out[3].present := FALSE;
   brand[14].out[3].byteOff := 0;
   brand[14].out[3].bitOff := 0;
   brand[14].out[3].inverted := FALSE;
   brand[14].out[4].present := FALSE;
   brand[14].out[4].byteOff := 0;
   brand[14].out[4].bitOff := 0;
   brand[14].out[4].inverted := FALSE;
   brand[14].out[5].present := FALSE;
   brand[14].out[5].byteOff := 0;
   brand[14].out[5].bitOff := 0;
   brand[14].out[5].inverted := FALSE;
   brand[14].out[6].present := FALSE;
   brand[14].out[6].byteOff := 0;
   brand[14].out[6].bitOff := 0;
   brand[14].out[6].inverted := FALSE;
   brand[14].out[7].present := FALSE;
   brand[14].out[7].byteOff := 0;
   brand[14].out[7].bitOff := 0;
   brand[14].out[7].inverted := FALSE;
   brand[14].out[8].present := FALSE;
   brand[14].out[8].byteOff := 0;
   brand[14].out[8].bitOff := 0;
   brand[14].out[8].inverted := FALSE;
   brand[14].out[9].present := FALSE;
   brand[14].out[9].byteOff := 0;
   brand[14].out[9].bitOff := 0;
   brand[14].out[9].inverted := FALSE;
   brand[14].out[10].present := FALSE;
   brand[14].out[10].byteOff := 0;
   brand[14].out[10].bitOff := 0;
   brand[14].out[10].inverted := FALSE;
   brand[15]."name" := '';
   brand[15].cycleArchetype := 0;
   brand[15].in[0].present := FALSE;
   brand[15].in[0].byteOff := 0;
   brand[15].in[0].bitOff := 0;
   brand[15].in[0].inverted := FALSE;
   brand[15].in[1].present := FALSE;
   brand[15].in[1].byteOff := 0;
   brand[15].in[1].bitOff := 0;
   brand[15].in[1].inverted := FALSE;
   brand[15].in[2].present := FALSE;
   brand[15].in[2].byteOff := 0;
   brand[15].in[2].bitOff := 0;
   brand[15].in[2].inverted := FALSE;
   brand[15].in[3].present := FALSE;
   brand[15].in[3].byteOff := 0;
   brand[15].in[3].bitOff := 0;
   brand[15].in[3].inverted := FALSE;
   brand[15].in[4].present := FALSE;
   brand[15].in[4].byteOff := 0;
   brand[15].in[4].bitOff := 0;
   brand[15].in[4].inverted := FALSE;
   brand[15].in[5].present := FALSE;
   brand[15].in[5].byteOff := 0;
   brand[15].in[5].bitOff := 0;
   brand[15].in[5].inverted := FALSE;
   brand[15].in[6].present := FALSE;
   brand[15].in[6].byteOff := 0;
   brand[15].in[6].bitOff := 0;
   brand[15].in[6].inverted := FALSE;
   brand[15].in[7].present := FALSE;
   brand[15].in[7].byteOff := 0;
   brand[15].in[7].bitOff := 0;
   brand[15].in[7].inverted := FALSE;
   brand[15].in[8].present := FALSE;
   brand[15].in[8].byteOff := 0;
   brand[15].in[8].bitOff := 0;
   brand[15].in[8].inverted := FALSE;
   brand[15].in[9].present := FALSE;
   brand[15].in[9].byteOff := 0;
   brand[15].in[9].bitOff := 0;
   brand[15].in[9].inverted := FALSE;
   brand[15].out[0].present := FALSE;
   brand[15].out[0].byteOff := 0;
   brand[15].out[0].bitOff := 0;
   brand[15].out[0].inverted := FALSE;
   brand[15].out[1].present := FALSE;
   brand[15].out[1].byteOff := 0;
   brand[15].out[1].bitOff := 0;
   brand[15].out[1].inverted := FALSE;
   brand[15].out[2].present := FALSE;
   brand[15].out[2].byteOff := 0;
   brand[15].out[2].bitOff := 0;
   brand[15].out[2].inverted := FALSE;
   brand[15].out[3].present := FALSE;
   brand[15].out[3].byteOff := 0;
   brand[15].out[3].bitOff := 0;
   brand[15].out[3].inverted := FALSE;
   brand[15].out[4].present := FALSE;
   brand[15].out[4].byteOff := 0;
   brand[15].out[4].bitOff := 0;
   brand[15].out[4].inverted := FALSE;
   brand[15].out[5].present := FALSE;
   brand[15].out[5].byteOff := 0;
   brand[15].out[5].bitOff := 0;
   brand[15].out[5].inverted := FALSE;
   brand[15].out[6].present := FALSE;
   brand[15].out[6].byteOff := 0;
   brand[15].out[6].bitOff := 0;
   brand[15].out[6].inverted := FALSE;
   brand[15].out[7].present := FALSE;
   brand[15].out[7].byteOff := 0;
   brand[15].out[7].bitOff := 0;
   brand[15].out[7].inverted := FALSE;
   brand[15].out[8].present := FALSE;
   brand[15].out[8].byteOff := 0;
   brand[15].out[8].bitOff := 0;
   brand[15].out[8].inverted := FALSE;
   brand[15].out[9].present := FALSE;
   brand[15].out[9].byteOff := 0;
   brand[15].out[9].bitOff := 0;
   brand[15].out[9].inverted := FALSE;
   brand[15].out[10].present := FALSE;
   brand[15].out[10].byteOff := 0;
   brand[15].out[10].bitOff := 0;
   brand[15].out[10].inverted := FALSE;
   brand[16]."name" := '';
   brand[16].cycleArchetype := 0;
   brand[16].in[0].present := FALSE;
   brand[16].in[0].byteOff := 0;
   brand[16].in[0].bitOff := 0;
   brand[16].in[0].inverted := FALSE;
   brand[16].in[1].present := FALSE;
   brand[16].in[1].byteOff := 0;
   brand[16].in[1].bitOff := 0;
   brand[16].in[1].inverted := FALSE;
   brand[16].in[2].present := FALSE;
   brand[16].in[2].byteOff := 0;
   brand[16].in[2].bitOff := 0;
   brand[16].in[2].inverted := FALSE;
   brand[16].in[3].present := FALSE;
   brand[16].in[3].byteOff := 0;
   brand[16].in[3].bitOff := 0;
   brand[16].in[3].inverted := FALSE;
   brand[16].in[4].present := FALSE;
   brand[16].in[4].byteOff := 0;
   brand[16].in[4].bitOff := 0;
   brand[16].in[4].inverted := FALSE;
   brand[16].in[5].present := FALSE;
   brand[16].in[5].byteOff := 0;
   brand[16].in[5].bitOff := 0;
   brand[16].in[5].inverted := FALSE;
   brand[16].in[6].present := FALSE;
   brand[16].in[6].byteOff := 0;
   brand[16].in[6].bitOff := 0;
   brand[16].in[6].inverted := FALSE;
   brand[16].in[7].present := FALSE;
   brand[16].in[7].byteOff := 0;
   brand[16].in[7].bitOff := 0;
   brand[16].in[7].inverted := FALSE;
   brand[16].in[8].present := FALSE;
   brand[16].in[8].byteOff := 0;
   brand[16].in[8].bitOff := 0;
   brand[16].in[8].inverted := FALSE;
   brand[16].in[9].present := FALSE;
   brand[16].in[9].byteOff := 0;
   brand[16].in[9].bitOff := 0;
   brand[16].in[9].inverted := FALSE;
   brand[16].out[0].present := FALSE;
   brand[16].out[0].byteOff := 0;
   brand[16].out[0].bitOff := 0;
   brand[16].out[0].inverted := FALSE;
   brand[16].out[1].present := FALSE;
   brand[16].out[1].byteOff := 0;
   brand[16].out[1].bitOff := 0;
   brand[16].out[1].inverted := FALSE;
   brand[16].out[2].present := FALSE;
   brand[16].out[2].byteOff := 0;
   brand[16].out[2].bitOff := 0;
   brand[16].out[2].inverted := FALSE;
   brand[16].out[3].present := FALSE;
   brand[16].out[3].byteOff := 0;
   brand[16].out[3].bitOff := 0;
   brand[16].out[3].inverted := FALSE;
   brand[16].out[4].present := FALSE;
   brand[16].out[4].byteOff := 0;
   brand[16].out[4].bitOff := 0;
   brand[16].out[4].inverted := FALSE;
   brand[16].out[5].present := FALSE;
   brand[16].out[5].byteOff := 0;
   brand[16].out[5].bitOff := 0;
   brand[16].out[5].inverted := FALSE;
   brand[16].out[6].present := FALSE;
   brand[16].out[6].byteOff := 0;
   brand[16].out[6].bitOff := 0;
   brand[16].out[6].inverted := FALSE;
   brand[16].out[7].present := FALSE;
   brand[16].out[7].byteOff := 0;
   brand[16].out[7].bitOff := 0;
   brand[16].out[7].inverted := FALSE;
   brand[16].out[8].present := FALSE;
   brand[16].out[8].byteOff := 0;
   brand[16].out[8].bitOff := 0;
   brand[16].out[8].inverted := FALSE;
   brand[16].out[9].present := FALSE;
   brand[16].out[9].byteOff := 0;
   brand[16].out[9].bitOff := 0;
   brand[16].out[9].inverted := FALSE;
   brand[16].out[10].present := FALSE;
   brand[16].out[10].byteOff := 0;
   brand[16].out[10].bitOff := 0;
   brand[16].out[10].inverted := FALSE;

END_DATA_BLOCK

